// TIA Portal V19 export
FUNCTION "FC_Search_HW" : Void   // FC14, STL
TITLE = ermittelt ggf. HW-Pos
{ S7_Optimized_Access := 'FALSE' }
AUTHOR : MS
// sucht in Fahrtrichtung nach einem notwendigen Höhenwechsel
// und gibt die Höhenwechselposition und die Zielebene zurück
// stored: AutoNumber false
   VAR_INPUT
      SO_li : Bool;   // Sensor Oben aktiv --> kein HW notwendig
      SO_re : Bool;   // Sensor Oben aktiv --> kein HW notwendig
   END_VAR
   VAR_IN_OUT
      IstPos : DInt;   // Istposition des FW in Inkrementen
      ZielPos : DInt;   // Position an der ein Höhenwechsel erfolgt (ohne HW:=tmp.FW_ZIEL_POS)
      Bereich_Ziel : DInt;   // Zielbereich für Positionierung
      Bereich_langsam : DInt;   // Bereich für Langsamfahrt
      FW_Ebene_li : Byte;   // aktuelle FW-Ebene
      Zielebene_li : Byte;   // Ebene die FW im Ziel einnehmen soll
      HW_akt_li : Bool;   // ist dieses Bit gesetzt wurde bereits eine HW-Pos ermittelt
      FW_Ebene_re : Byte;   // aktuelle FW-Ebene
      Zielebene_re : Byte;   // Ebene die FW im Ziel einnehmen soll
      HW_akt_re : Bool;   // ist dieses Bit gesetzt wurde bereits eine HW-Pos ermittelt
   END_VAR
   VAR_TEMP
      count : Int;   // Loopcounter
      fwd : Bool;   // FW bewegt sich in Richtung höhere Position
      HW_Mitte : Bool;   // Höhenwechselposition erreicht
      HW_Pos : DInt;   // an dieser Stelle gilt eine andere Ebene
   END_VAR
BEGIN

NETWORK
TITLE = Initialisierung
// Ist kein Höhenwechsel notwendig wird die aktuelle FW-Ebene als Zielebene und 
// die 
// Tmp.FW_ZIEL_POS als Ziel zurückgegeben.
//Initialisierung
      L     #FW_Ebene_li;
      T     #Zielebene_li;
      L     #FW_Ebene_re;
      T     #Zielebene_re;

      A     #SO_li;
      A     #SO_re;
//existiert ein Höhenwechsel
      ON    "DB_ANLAGE".config.HW_exist;
      R     #HW_akt_li;
      R     #HW_akt_re;
      BEC;

      L     #ZielPos;
      L     #IstPos;
      >D;
      =     #fwd;


NETWORK
TITLE = Scanning
// Suche nach HW-Pos
//FW hat Ziel bereits erreicht
      L     #ZielPos;
      L     #Bereich_Ziel;
      -D;
      L     #IstPos;
      >D;
      JC    chk;
      L     #ZielPos;
      L     #Bereich_Ziel;
      +D;
      L     #IstPos;
      <D;
      JC    chk;
      BE;

chk:  L     0;
retH: T     #count;
      L     "DB_HW".Anzahl;  //HW-Eintrag Länge
      >=I;
      BEC;
      A     #fwd;
      L     #count;
      JC    fwdH;
      +     1;
      -I;
fwdH: L     "DB_HW".lengHW;  //HW-Eintrag Länge
      *I;
      L     "DB_HW".Offset;  //HW-Einträge Offset
      +I;
      SLD   3;
      LAR2;
      OPN   "DB_HW";
      L     0;
      L     DBD [AR2, P#0.0];  //"DB_HW".HW[x].Pos
      ==D;
      BEC;
//HW Mitte?
      L     DBD [AR2, P#0.0];  //"DB_HW".HW[x].Pos
      L     #IstPos;
      -D;
      DTR;
      ABS;
      RND;
      L     #Bereich_Ziel;
      <=D;
      =     #HW_Mitte;
      JC    fnd;

      A     #fwd;
      JC    vor;

//FW hat HW-Pos bereits hinter sich
      L     #IstPos;
      L     DBD [AR2, P#0.0];  //"DB_HW".HW[x].Pos
      <=D;
      JC    nexH;
//Ziel liegt noch vor HW
      L     #ZielPos;
      L     DBD [AR2, P#0.0];  //"DB_HW".HW[x].Pos
      >=D;
      BEC;
//Höhenwechsel liegt auf dem Weg
      JU    fnd;  //Höhenwechel gefunden

vor:  NOP   0;
//FW hat HW-Pos bereits hinter sich
      L     #IstPos;
      L     DBD [AR2, P#0.0];  //"DB_HW".HW[x].Pos
      >=D;
      JC    nexH;
//Ziel liegt noch vor HW
      L     #ZielPos;
      L     DBD [AR2, P#0.0];  //"DB_HW".HW[x].Pos
      <=D;
      BEC;
//Höhenwechsel liegt auf dem Weg
      JU    fnd;  //Höhenwechel gefunden

nexH: L     #count;
      L     1;
      +I;
      JU    retH;

//HW-gefunden
fnd:  A     #SO_li;
      JC    fnd_re;
      A     #fwd;
      JC    fwrd;
      L     DBB [AR2, P#4.0];  //"DB_HW".HW[x].Ebene_rck
      T     #Zielebene_li;
      JU    HWT;
fwrd: L     DBB [AR2, P#5.0];  //"DB_HW".HW[x].Ebene_vor
      T     #Zielebene_li;
HWT:  L     #FW_Ebene_li;
      ==I;
      JC    fnd_re;
      S     #HW_akt_li;
      L     DBD [AR2, P#0.0];  //"DB_HW".HW[x].Pos
      T     #ZielPos;

fnd_re:A     #SO_re;
      BEC;
      A     #fwd;
      JC    fwrd_re;
      L     DBB [AR2, P#4.0];  //"DB_HW".HW[x].Ebene_rck
      T     #Zielebene_re;
      JU    HWT_re;
fwrd_re:L     DBB [AR2, P#5.0];  //"DB_HW".HW[x].Ebene_vor
      T     #Zielebene_re;
HWT_re:L     #FW_Ebene_re;
      ==I;
      BEC;
      S     #HW_akt_re;
      L     DBD [AR2, P#0.0];  //"DB_HW".HW[x].Pos
      T     #ZielPos;
      BE;

END_FUNCTION
